TYPE ST_GROUP_STATE :
STRUCT
  State           : E_GROUP_STATE;
  McState         : MC_GROUP_STATE;
  AxisCount       : UINT;
END_STRUCT
END_TYPE

(* stored: Version 1.1.0.1, ProductVersion 3.1.4024.12
   DUT ST_GROUP_STATE: Id {432d19ce-aa25-4d8c-91c2-3d57f138f617} *)
